{attribute addProperty BoxType "EL2014-0000-0016"}
{attribute addProperty Id "ChannelAT %Q*ARRAY[0 ..3] OF Channel_D3FEAEF940.50"}
{attribute addProperty CRC "1283853898"}
{attribute addProperty SizeInBites "4"}
{attribute addProperty SizeInBytes "0.5"}
TYPE DIG_Outputs_276DFED3 :
STRUCT
	{attribute addProperty Name "Channel"}
	Channel AT %Q* : ARRAY[0 ..3] OF Channel_D3FEAEF9;
END_STRUCT
END_TYPE

(* stored: Version 1.2.0.0, ProductVersion 3.1.4024.9
   DUT DIG_Outputs_276DFED3: Id {5133e165-b8f2-488b-8e77-2fbbd50d1bb8} *)
